Omron CX-Programmer project NewProject (CX-Programmer 9.73)

# PLC NewPLC1: CP1E N30

## Program NewProgram1 (cyclic task 0)

### Section Section1

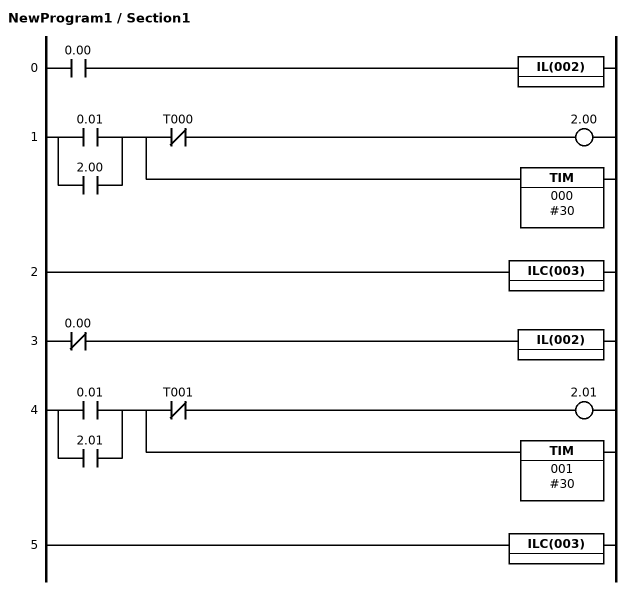
; rung 0
LD 0.00
IL(002)
; rung 1
LD 0.01
OR 2.00
OUT TR0
ANDNOT T000
OUT 2.00
LD TR0
TIM 000 #30
; rung 2
ILC(003)
; rung 3
LDNOT 0.00
IL(002)
; rung 4
LD 0.01
OR 2.01
OUT TR0
ANDNOT T001
OUT 2.01
LD TR0
TIM 001 #30
; rung 5
ILC(003)

### Section END
; rung 0
END(001)